(* Schneider Machine Expert - Basic project PLC1, file version 2.7.0.0 *)
(* CompanyInformations: Name=Saxion *)
(* ProjectInformations: Name=TPAC - LFT Handling *)

HARDWARE
  Cpu 0: TM221CE24T
  EthernetConfiguration: NetworkName=M221, IpAllocationMode=FixedAddress, IpAddress=10.10.120.250, SubnetMask=255.255.255.0
  SerialLineConfiguration: Baud=Baud19200, Parity=ParityEven, DataBits=DataBits8, StopBits=StopBits1, PhysicalMedium=PhysicalMediumRs485, SlaveId=1, Addressing=SlaveAddressing
  MastTask: UsePeriodScanMode=false, PeriodScan=100
  FastTask: Period=255
  CpuBehavior: StartingMode=StartAsPreviousState, AutoSaveRamOnEeprom=true, WatchdogPeriod=250

SYMBOLS  (address, symbol, comment, settings)
  %M10      ALWAYS_FALSE
  %M11      ALWAYS_TRUE
  %M20      INC_TRANSBAAN
  %M30      STAP10ACTIVEER
  %M50      B_SAFETYOK
  %M51      RUN_AUTO
  %M52      RUN_RESET
  %M53      STOP
  %M54      RUN_PRG_TEST
  %M55      RUN_PRG
  %M56      RUN_TRANSBAAN
  %M57      RUN_SIM
  %M60      KUKASTART9
  %M61      KUKASTART10
  %M62      KUKASTART11
  %M63      KUKASTART_SPARE
  %M64      KUKASTART_SPARE1
  %M65      KUKASTOP_1
  %M66      KUKASTOP_2
  %M67      KUKASTOP_3
  %M68      QX_VENTIEL1
  %M69      QX_VENTIEL2
  %M70      QX_VENTIEL3
  %M80      QX_RELAISEXSTART
  %M81      QX_RELAISEXSTOP
  %M84      QX_VENTIEL1  "Start eindbeweging"
  %M85      QX_CUTTINGTOOLACTIVEER
  %M86      QX_CUTTINGTOOLDEACTIVEER
  %M98      QX_STARTTRANSBAAN
  %M99      QX_STOPTRANSBAAN
  %M100     IX_STARTKNOP
  %M101     IX_STOPKNOP
  %M102     IX_ESTOP
  %M103     IX_FCLENGTE
  %M104     IX_FCGRIPPER
  %M105     IX_REEDCUTTINGOPEN
  %M106     IX_REEDCUTTINGGESLOTEN
  %M107     IX_REEDGRIPPER1
  %M108     IX_REEDGRIPPER2
  %M109     IX_KUKAGEREED
  %M110     IX_KUKAALARM
  %M111     IX_KUKATUSSEN
  %M112     IX_CUTTERHAND
  %M120     IX_RESET
  %MW10     PRG_STAPPEN
  %MW12     ALARMCODE_PRG
  %TM1      T_STAP1  [Preset=2, Base=OneSecond]
  %TM2      T_STAP2  [Preset=2, Base=OneSecond]
  %TM3      T_ALARMSTAP2  "Timeout voor alarm"  [Preset=60, Base=OneSecond]
  %TM4      T_ALARMSTAP4  [Preset=5, Base=OneSecond]
  %TM5      T_ALARMSTAP5  [Preset=5, Base=OneSecond]
  %TM6      T_WACHTNACUT  [Preset=2, Base=OneSecond]
  %TM7      T_ALARMSTAP7  [Preset=30, Base=OneSecond]
  %TM8      T_STAP7  [Preset=2, Base=OneSecond]
  %TM9      T_ALARMSTAP8  [Preset=10, Base=OneSecond]
  %TM10     T_STAP9  [Preset=2, Base=OneSecond]
  %TM11     T_ALARMSTAP10  [Preset=10, Base=OneSecond]
  %TM12     T_STAP10  [Type=TP, Preset=3, Base=OneSecond]
  %TM13     T_STAP11  [Preset=3, Base=OneSecond]
  %TM14     T_ALARMSTAP11  [Preset=10, Base=OneSecond]
  %TM20     T_STARTKNOP  [Preset=1, Base=OneSecond]
  %TM21     T_STOPKNOP  [Preset=1, Base=OneSecond]
  %TM66       [Preset=30, Base=OneSecond]
  %I0.0     PB01
  %I0.1     PB02
  %I0.2     PB03
  %I0.3     FC01
  %I0.4     FC02
  %I0.5     RC01
  %I0.6     RC02
  %I0.7     RG01
  %I0.8     RG02
  %I0.9     IKS01
  %I0.10    IKS02
  %I0.11    IKS03
  %I0.12    PB04

POU ALIAS
  (* SectionNumber=1 *)

// Rung 0
  LD 1                    (* Alias POU regelt in/uitgangen *)
  ST %M11                 (* ALWAYS_TRUE - Zet simuleer bit %M57 om hardware I/O inactief te zetten. *)
  STN %M10                (* ALWAYS_FALSE *)
  // as ST:
  //   ALWAYS_TRUE := TRUE;
  //   ALWAYS_FALSE := FALSE;

// Rung 1: Startknop
  BLK %TM20               (* T_STARTKNOP *)
  LD %I0.0                (* PB01 *)
  ANDN %M57               (* RUN_SIM *)
  ANDN %M120              (* IX_RESET *)
  IN
  OUT_BLK
  LD Q
  ST %M100                (* IX_STARTKNOP *)
  END_BLK
  // as ST:
  //   T_STARTKNOP(IN := PB01 AND NOT RUN_SIM AND NOT IX_RESET);
  //   IX_STARTKNOP := T_STARTKNOP.Q;

// Rung 2: Stopknop
  BLK %TM21               (* T_STOPKNOP *)
  LD %I0.1                (* PB02 *)
  ANDN %M57               (* RUN_SIM *)
  ANDN %M120              (* IX_RESET *)
  IN
  OUT_BLK
  LD Q
  ST %M101                (* IX_STOPKNOP *)
  END_BLK
  // as ST:
  //   T_STOPKNOP(IN := PB02 AND NOT RUN_SIM AND NOT IX_RESET);
  //   IX_STOPKNOP := T_STOPKNOP.Q;

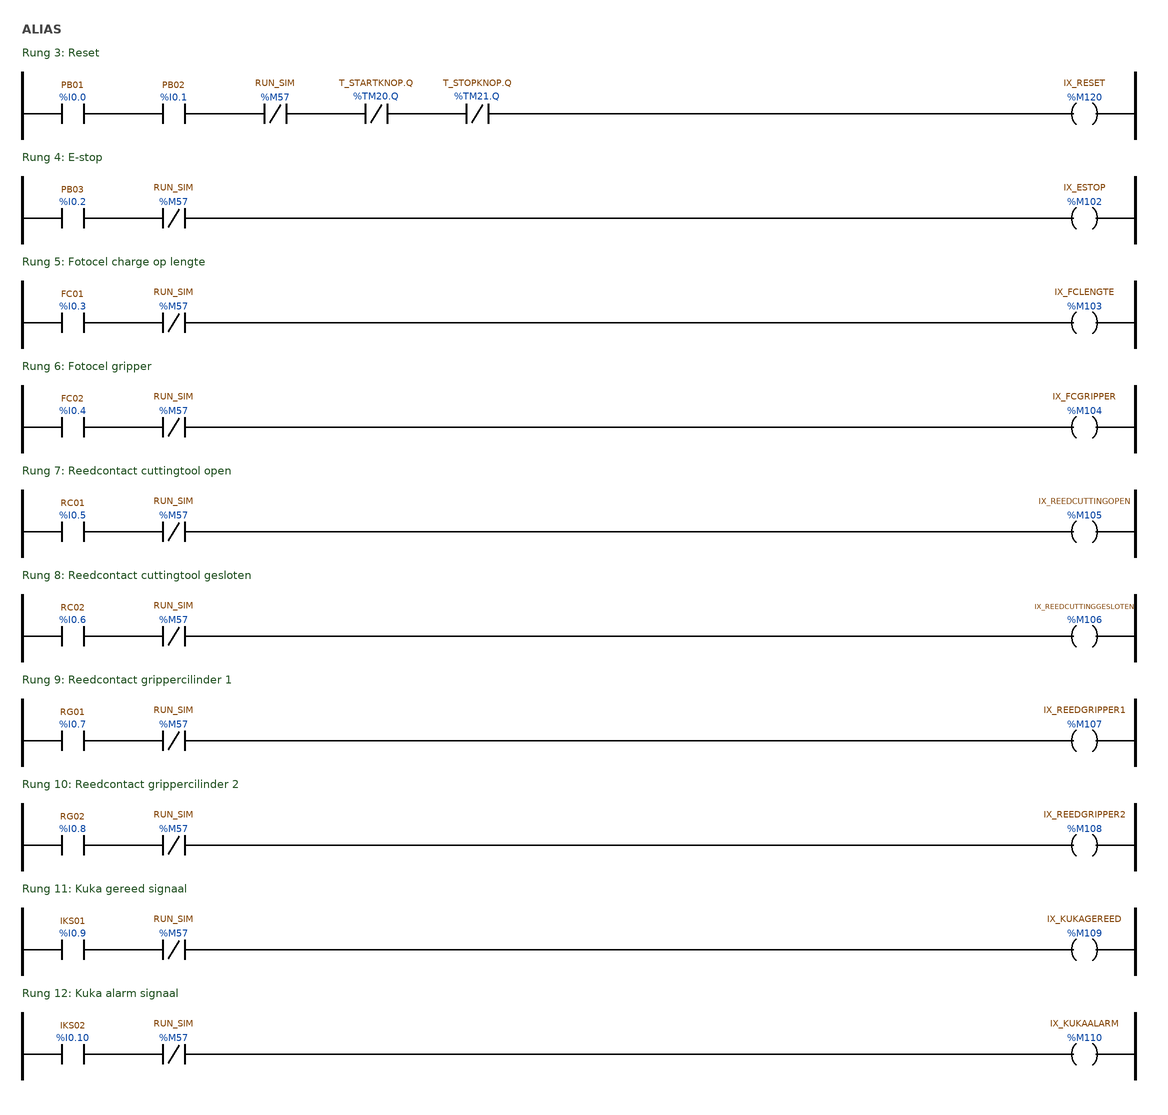

// Rung 3: Reset
  LD %I0.0                (* PB01 *)
  AND %I0.1               (* PB02 *)
  ANDN %M57               (* RUN_SIM *)
  ANDN %TM20.Q            (* T_STARTKNOP *)
  ANDN %TM21.Q            (* T_STOPKNOP *)
  ST %M120                (* IX_RESET *)
  // as ST:
  //   IX_RESET := PB01 AND PB02 AND NOT RUN_SIM AND NOT T_STARTKNOP.Q AND NOT T_STOPKNOP.Q;

// Rung 4: E-stop
  LD %I0.2                (* PB03 *)
  ANDN %M57               (* RUN_SIM *)
  ST %M102                (* IX_ESTOP *)
  // as ST:
  //   IX_ESTOP := PB03 AND NOT RUN_SIM;

// Rung 5: Fotocel charge op lengte
  LD %I0.3                (* FC01 *)
  ANDN %M57               (* RUN_SIM *)
  ST %M103                (* IX_FCLENGTE *)
  // as ST:
  //   IX_FCLENGTE := FC01 AND NOT RUN_SIM;

// Rung 6: Fotocel gripper
  LD %I0.4                (* FC02 *)
  ANDN %M57               (* RUN_SIM *)
  ST %M104                (* IX_FCGRIPPER *)
  // as ST:
  //   IX_FCGRIPPER := FC02 AND NOT RUN_SIM;

// Rung 7: Reedcontact cuttingtool open
  LD %I0.5                (* RC01 *)
  ANDN %M57               (* RUN_SIM *)
  ST %M105                (* IX_REEDCUTTINGOPEN *)
  // as ST:
  //   IX_REEDCUTTINGOPEN := RC01 AND NOT RUN_SIM;

// Rung 8: Reedcontact cuttingtool gesloten
  LD %I0.6                (* RC02 *)
  ANDN %M57               (* RUN_SIM *)
  ST %M106                (* IX_REEDCUTTINGGESLOTEN *)
  // as ST:
  //   IX_REEDCUTTINGGESLOTEN := RC02 AND NOT RUN_SIM;

// Rung 9: Reedcontact grippercilinder 1
  LD %I0.7                (* RG01 *)
  ANDN %M57               (* RUN_SIM *)
  ST %M107                (* IX_REEDGRIPPER1 *)
  // as ST:
  //   IX_REEDGRIPPER1 := RG01 AND NOT RUN_SIM;

// Rung 10: Reedcontact grippercilinder 2
  LD %I0.8                (* RG02 *)
  ANDN %M57               (* RUN_SIM *)
  ST %M108                (* IX_REEDGRIPPER2 *)
  // as ST:
  //   IX_REEDGRIPPER2 := RG02 AND NOT RUN_SIM;

// Rung 11: Kuka gereed signaal
  LD %I0.9                (* IKS01 *)
  ANDN %M57               (* RUN_SIM *)
  ST %M109                (* IX_KUKAGEREED *)
  // as ST:
  //   IX_KUKAGEREED := IKS01 AND NOT RUN_SIM;

// Rung 12: Kuka alarm signaal
  LD %I0.10               (* IKS02 *)
  ANDN %M57               (* RUN_SIM *)
  ST %M110                (* IX_KUKAALARM *)
  // as ST:
  //   IX_KUKAALARM := IKS02 AND NOT RUN_SIM;

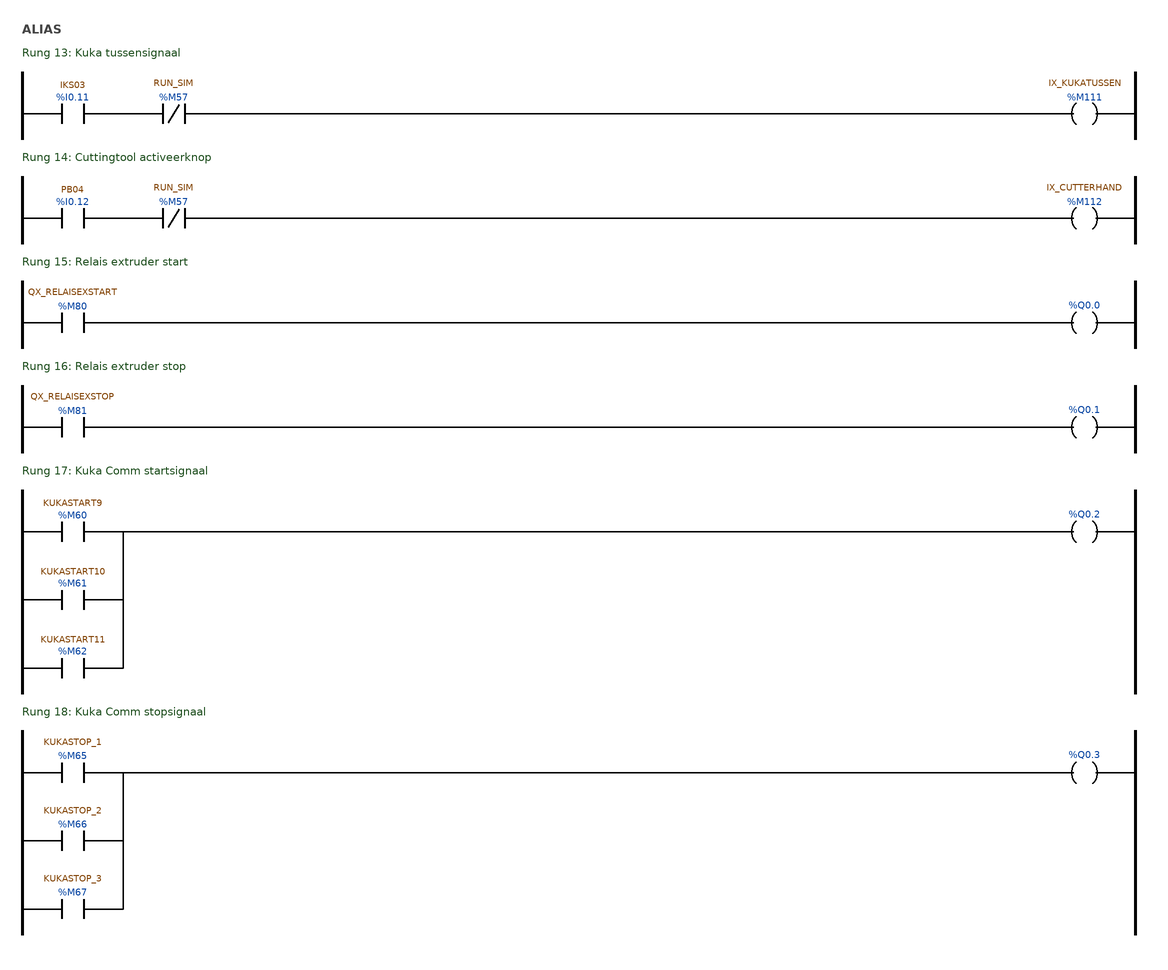

// Rung 13: Kuka tussensignaal
  LD %I0.11               (* IKS03 *)
  ANDN %M57               (* RUN_SIM *)
  ST %M111                (* IX_KUKATUSSEN *)
  // as ST:
  //   IX_KUKATUSSEN := IKS03 AND NOT RUN_SIM;

// Rung 14: Cuttingtool activeerknop
  LD %I0.12               (* PB04 *)
  ANDN %M57               (* RUN_SIM *)
  ST %M112                (* IX_CUTTERHAND *)
  // as ST:
  //   IX_CUTTERHAND := PB04 AND NOT RUN_SIM;

// Rung 15: Relais extruder start
  LD %M80                 (* QX_RELAISEXSTART *)
  ST %Q0.0
  // as ST:
  //   %Q0.0 := QX_RELAISEXSTART;

// Rung 16: Relais extruder stop
  LD %M81                 (* QX_RELAISEXSTOP *)
  ST %Q0.1
  // as ST:
  //   %Q0.1 := QX_RELAISEXSTOP;

// Rung 17: Kuka Comm startsignaal
  LD %M60                 (* KUKASTART9 *)
  OR %M61                 (* KUKASTART10 *)
  OR %M62                 (* KUKASTART11 *)
  ST %Q0.2
  // as ST:
  //   %Q0.2 := KUKASTART9 OR KUKASTART10 OR KUKASTART11;

// Rung 18: Kuka Comm stopsignaal
  LD %M65                 (* KUKASTOP_1 *)
  OR %M66                 (* KUKASTOP_2 *)
  OR %M67                 (* KUKASTOP_3 *)
  ST %Q0.3
  // as ST:
  //   %Q0.3 := KUKASTOP_1 OR KUKASTOP_2 OR KUKASTOP_3;

// Rung 19: Ventiel1/Kuka Alarmsignaal
  LD %M68                 (* QX_VENTIEL1 *)
  ST %Q0.4
  // as ST:
  //   %Q0.4 := QX_VENTIEL1;

// Rung 20
  LD %M85                 (* QX_CUTTINGTOOLACTIVEER *)
  ST %Q0.5
  // as ST:
  //   %Q0.5 := QX_CUTTINGTOOLACTIVEER;

// Rung 21
  LD %M86                 (* QX_CUTTINGTOOLDEACTIVEER *)
  ST %Q0.6
  // as ST:
  //   %Q0.6 := QX_CUTTINGTOOLDEACTIVEER;

POU Safety
  (* SectionNumber=2 *)

// Rung 22: Lees ingangen
  LD %M102                (* IX_ESTOP - // Laad E-STOP signal (NC) *)
  ANDN %M110              (* IX_KUKAALARM - // KUKA Alarm Signal (NO) *)
  ST %M50                 (* B_SAFETYOK - // Zet resultaat in safety bit *)
  // as ST:
  //   B_SAFETYOK := IX_ESTOP AND NOT IX_KUKAALARM;

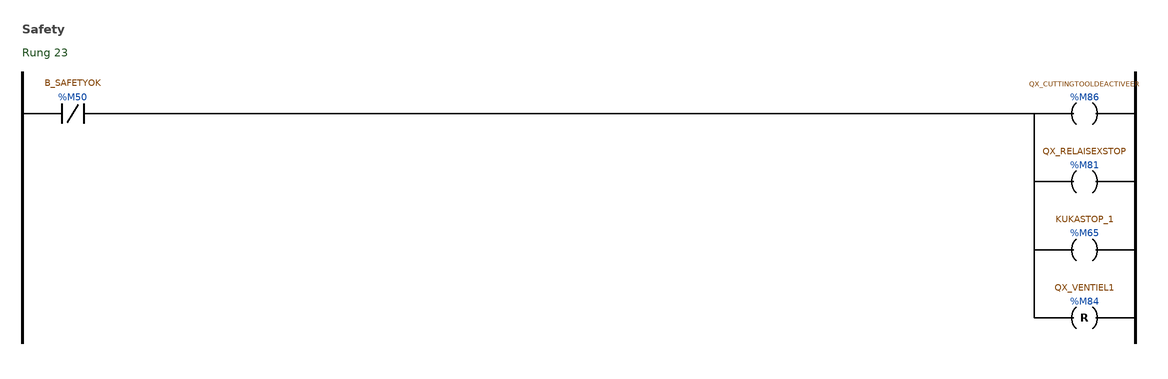

// Rung 23
  LDN %M50                (* B_SAFETYOK *)
  ST %M86                 (* QX_CUTTINGTOOLDEACTIVEER *)
  ST %M81                 (* QX_RELAISEXSTOP *)
  ST %M65                 (* KUKASTOP_1 *)
  R %M84                  (* QX_VENTIEL1 *)
  // as ST:
  //   QX_CUTTINGTOOLDEACTIVEER := NOT B_SAFETYOK;
  //   QX_RELAISEXSTOP := NOT B_SAFETYOK;
  //   KUKASTOP_1 := NOT B_SAFETYOK;
  //   IF NOT B_SAFETYOK THEN QX_VENTIEL1 := FALSE; END_IF;

POU Modus
  (* SectionNumber=3 *)

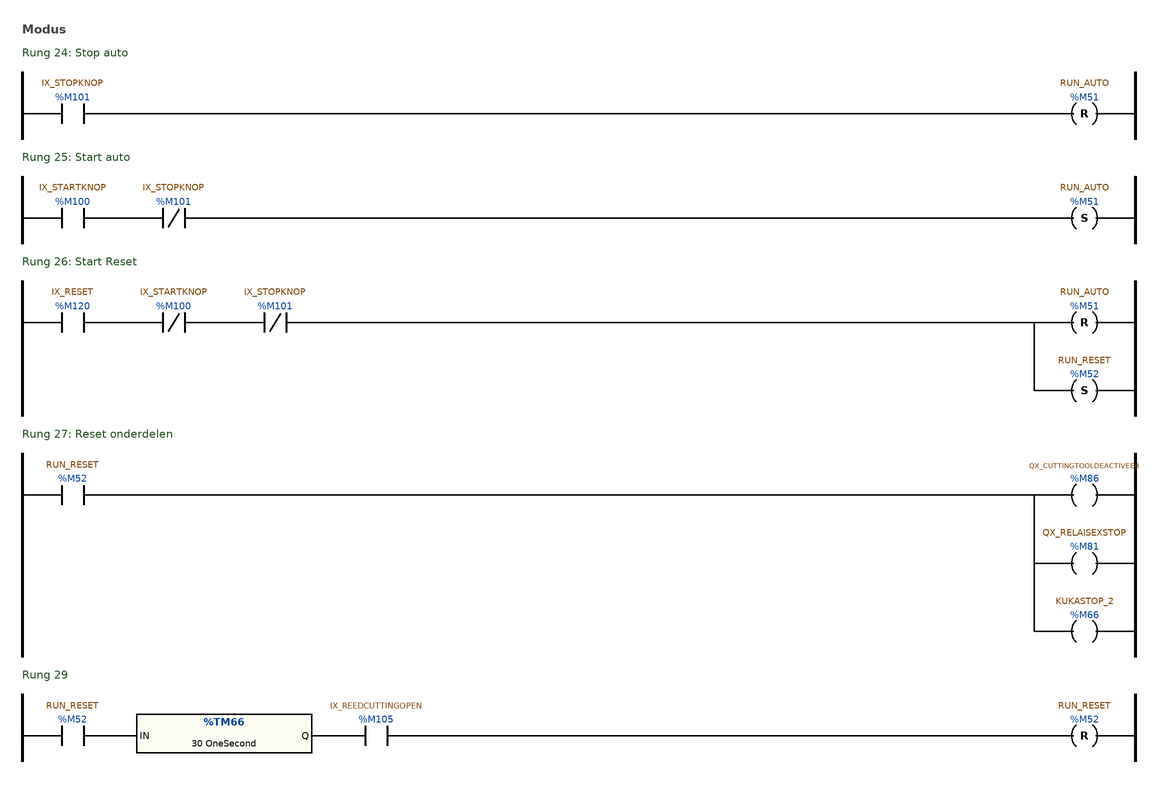

// Rung 24: Stop auto
  LD %M101                (* IX_STOPKNOP *)
  R %M51                  (* RUN_AUTO *)
  // as ST:
  //   IF IX_STOPKNOP THEN RUN_AUTO := FALSE; END_IF;

// Rung 25: Start auto
  LD %M100                (* IX_STARTKNOP *)
  ANDN %M101              (* IX_STOPKNOP *)
  S %M51                  (* RUN_AUTO *)
  // as ST:
  //   IF IX_STARTKNOP AND NOT IX_STOPKNOP THEN RUN_AUTO := TRUE; END_IF;

// Rung 26: Start Reset
  LD %M120                (* IX_RESET *)
  ANDN %M100              (* IX_STARTKNOP *)
  ANDN %M101              (* IX_STOPKNOP *)
  R %M51                  (* RUN_AUTO *)
  S %M52                  (* RUN_RESET *)
  // as ST:
  //   IF IX_RESET AND NOT IX_STARTKNOP AND NOT IX_STOPKNOP THEN RUN_AUTO := FALSE; END_IF;
  //   IF IX_RESET AND NOT IX_STARTKNOP AND NOT IX_STOPKNOP THEN RUN_RESET := TRUE; END_IF;

// Rung 27: Reset onderdelen
  LD %M52                 (* RUN_RESET *)
  ST %M86                 (* QX_CUTTINGTOOLDEACTIVEER *)
  ST %M81                 (* QX_RELAISEXSTOP *)
  ST %M66                 (* KUKASTOP_2 *)
  // as ST:
  //   QX_CUTTINGTOOLDEACTIVEER := RUN_RESET;
  //   QX_RELAISEXSTOP := RUN_RESET;
  //   KUKASTOP_2 := RUN_RESET;

// Rung 28: Reset programmastappen
// Res
  LD %M52                 (* RUN_RESET *)
  [ %MW10 := 0 ]          (* PRG_STAPPEN *)
  // as ST:
  //   IF RUN_RESET THEN PRG_STAPPEN := 0; END_IF;

// Rung 29
  BLK %TM66
  LD %M52                 (* RUN_RESET *)
  IN
  OUT_BLK
  LD Q
  AND %M105               (* IX_REEDCUTTINGOPEN *)
  R %M52                  (* RUN_RESET *)
  END_BLK
  // as ST:
  //   %TM66(IN := RUN_RESET);
  //   IF %TM66.Q AND IX_REEDCUTTINGOPEN THEN RUN_RESET := FALSE; END_IF;

POU PRG1
  (* SectionNumber=4 *)

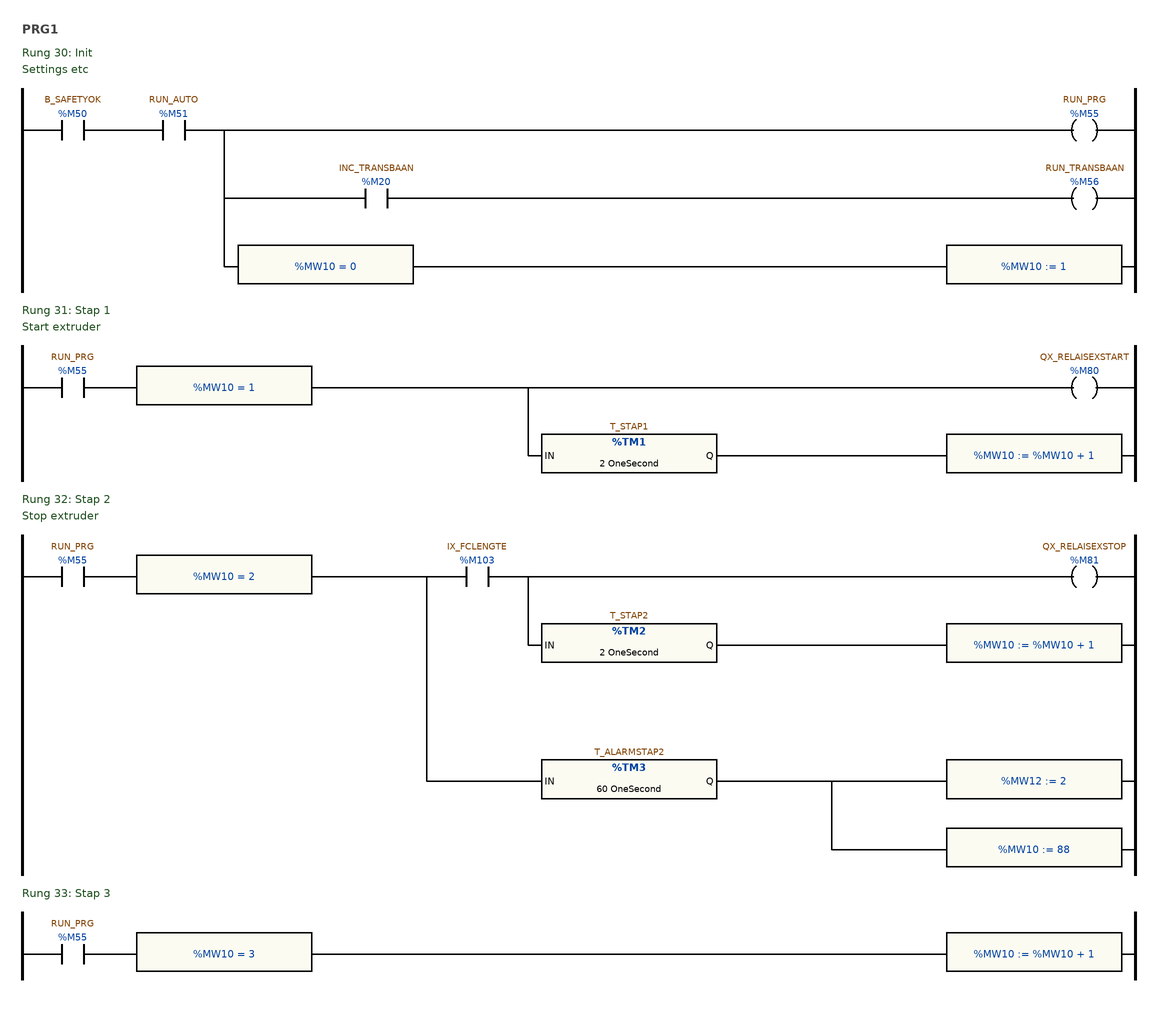

// Rung 30: Init
// Settings etc
  LD %M50                 (* B_SAFETYOK *)
  AND %M51                (* RUN_AUTO *)
  MPS
  ST %M55                 (* RUN_PRG *)
  MRD
  AND %M20                (* INC_TRANSBAAN *)
  ST %M56                 (* RUN_TRANSBAAN *)
  MPP
  AND [ %MW10 = 0 ]       (* PRG_STAPPEN *)
  [ %MW10 := 1 ]          (* PRG_STAPPEN *)
  // as ST:
  //   RUN_PRG := B_SAFETYOK AND RUN_AUTO;
  //   RUN_TRANSBAAN := B_SAFETYOK AND RUN_AUTO AND INC_TRANSBAAN;
  //   IF B_SAFETYOK AND RUN_AUTO AND PRG_STAPPEN = 0 THEN PRG_STAPPEN := 1; END_IF;

// Rung 31: Stap 1
// Start extruder
  LD 1
  MULTIFB
  LD 1
  AND %M55                (* RUN_PRG *)
  AND [ %MW10 = 1 ]       (* PRG_STAPPEN *)
  ST %MW2009:X0
  LD %MW2009:X0
  ST %M80                 (* QX_RELAISEXSTART *)
  BLK %TM1                (* T_STAP1 *)
  LD %MW2009:X0
  IN
  OUT_BLK
  LD Q
  [ %MW10 := %MW10 + 1 ]  (* PRG_STAPPEN, PRG_STAPPEN *)
  END_BLK
  MULTIFB
  // as ST:
  //   QX_RELAISEXSTART := RUN_PRG AND PRG_STAPPEN = 1;
  //   T_STAP1(IN := RUN_PRG AND PRG_STAPPEN = 1);
  //   IF T_STAP1.Q THEN PRG_STAPPEN := PRG_STAPPEN + 1; END_IF;

// Rung 32: Stap 2
// Stop extruder
  LD 1
  MULTIFB
  LD 1
  AND %M55                (* RUN_PRG *)
  AND [ %MW10 = 2 ]       (* PRG_STAPPEN *)
  ST %MW2009:X0
  LD %MW2009:X0
  AND %M103               (* IX_FCLENGTE *)
  ST %MW2009:X1
  LD %MW2009:X1
  ST %M81                 (* QX_RELAISEXSTOP *)
  BLK %TM2                (* T_STAP2 *)
  LD %MW2009:X1
  IN
  OUT_BLK
  LD Q
  [ %MW10 := %MW10 + 1 ]  (* PRG_STAPPEN, PRG_STAPPEN *)
  END_BLK
  BLK %TM3                (* T_ALARMSTAP2 *)
  LD %MW2009:X0
  IN
  OUT_BLK
  LD Q
  [ %MW12 := 2 ]          (* ALARMCODE_PRG *)
  [ %MW10 := 88 ]         (* PRG_STAPPEN *)
  END_BLK
  MULTIFB
  // as ST:
  //   QX_RELAISEXSTOP := RUN_PRG AND PRG_STAPPEN = 2 AND IX_FCLENGTE;
  //   T_STAP2(IN := RUN_PRG AND PRG_STAPPEN = 2 AND IX_FCLENGTE);
  //   _t1 := RUN_PRG AND PRG_STAPPEN = 2;
  //   IF T_STAP2.Q THEN PRG_STAPPEN := PRG_STAPPEN + 1; END_IF;
  //   T_ALARMSTAP2(IN := _t1);
  //   IF T_ALARMSTAP2.Q THEN ALARMCODE_PRG := 2; END_IF;
  //   IF T_ALARMSTAP2.Q THEN PRG_STAPPEN := 88; END_IF;

// Rung 33: Stap 3
  LD %M55                 (* RUN_PRG *)
  AND [ %MW10 = 3 ]       (* PRG_STAPPEN *)
  [ %MW10 := %MW10 + 1 ]  (* PRG_STAPPEN, PRG_STAPPEN *)
  // as ST:
  //   IF RUN_PRG AND PRG_STAPPEN = 3 THEN PRG_STAPPEN := PRG_STAPPEN + 1; END_IF;

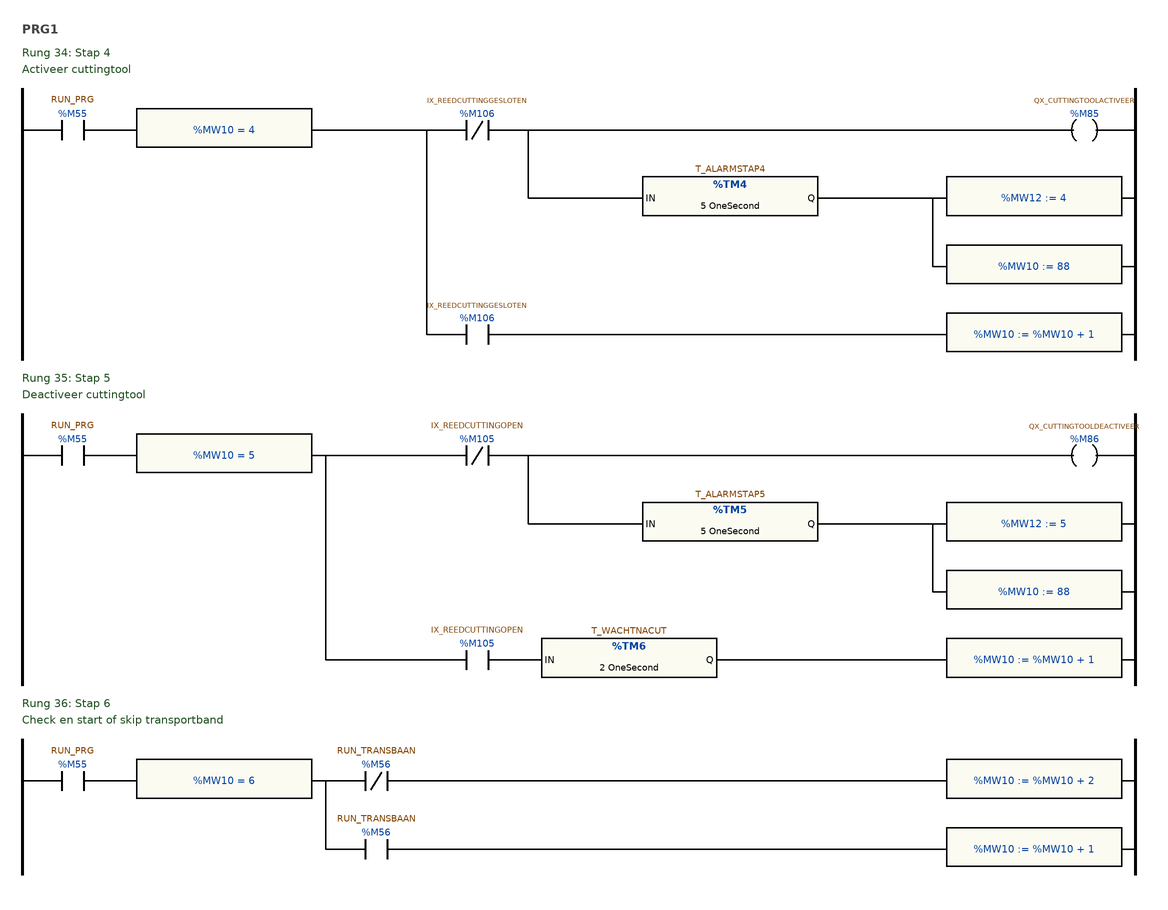

// Rung 34: Stap 4
// Activeer cuttingtool
  LD 1
  MULTIFB
  LD 1
  AND %M55                (* RUN_PRG *)
  AND [ %MW10 = 4 ]       (* PRG_STAPPEN *)
  ST %MW2009:X0
  LD %MW2009:X0
  ANDN %M106              (* IX_REEDCUTTINGGESLOTEN *)
  ST %MW2009:X1
  LD %MW2009:X1
  ST %M85                 (* QX_CUTTINGTOOLACTIVEER *)
  BLK %TM4                (* T_ALARMSTAP4 *)
  LD %MW2009:X1
  IN
  OUT_BLK
  LD Q
  [ %MW12 := 4 ]          (* ALARMCODE_PRG *)
  [ %MW10 := 88 ]         (* PRG_STAPPEN *)
  END_BLK
  LD %MW2009:X0
  AND %M106               (* IX_REEDCUTTINGGESLOTEN *)
  [ %MW10 := %MW10 + 1 ]  (* PRG_STAPPEN, PRG_STAPPEN *)
  MULTIFB
  // as ST:
  //   QX_CUTTINGTOOLACTIVEER := RUN_PRG AND PRG_STAPPEN = 4 AND NOT IX_REEDCUTTINGGESLOTEN;
  //   T_ALARMSTAP4(IN := RUN_PRG AND PRG_STAPPEN = 4 AND NOT IX_REEDCUTTINGGESLOTEN);
  //   IF T_ALARMSTAP4.Q THEN ALARMCODE_PRG := 4; END_IF;
  //   _t1 := RUN_PRG AND PRG_STAPPEN = 4;
  //   IF T_ALARMSTAP4.Q THEN PRG_STAPPEN := 88; END_IF;
  //   IF _t1 AND IX_REEDCUTTINGGESLOTEN THEN PRG_STAPPEN := PRG_STAPPEN + 1; END_IF;

// Rung 35: Stap 5
// Deactiveer cuttingtool
  LD 1
  MULTIFB
  LD 1
  AND %M55                (* RUN_PRG *)
  AND [ %MW10 = 5 ]       (* PRG_STAPPEN *)
  ST %MW2009:X0
  LD %MW2009:X0
  ANDN %M105              (* IX_REEDCUTTINGOPEN *)
  ST %MW2009:X1
  LD %MW2009:X1
  ST %M86                 (* QX_CUTTINGTOOLDEACTIVEER *)
  BLK %TM5                (* T_ALARMSTAP5 *)
  LD %MW2009:X1
  IN
  OUT_BLK
  LD Q
  [ %MW12 := 5 ]          (* ALARMCODE_PRG *)
  [ %MW10 := 88 ]         (* PRG_STAPPEN *)
  END_BLK
  BLK %TM6                (* T_WACHTNACUT *)
  LD %MW2009:X0
  AND %M105               (* IX_REEDCUTTINGOPEN *)
  IN
  OUT_BLK
  LD Q
  [ %MW10 := %MW10 + 1 ]  (* PRG_STAPPEN, PRG_STAPPEN *)
  END_BLK
  MULTIFB
  // as ST:
  //   QX_CUTTINGTOOLDEACTIVEER := RUN_PRG AND PRG_STAPPEN = 5 AND NOT IX_REEDCUTTINGOPEN;
  //   T_ALARMSTAP5(IN := RUN_PRG AND PRG_STAPPEN = 5 AND NOT IX_REEDCUTTINGOPEN);
  //   IF T_ALARMSTAP5.Q THEN ALARMCODE_PRG := 5; END_IF;
  //   _t1 := RUN_PRG AND PRG_STAPPEN = 5;
  //   IF T_ALARMSTAP5.Q THEN PRG_STAPPEN := 88; END_IF;
  //   T_WACHTNACUT(IN := _t1 AND IX_REEDCUTTINGOPEN);
  //   IF T_WACHTNACUT.Q THEN PRG_STAPPEN := PRG_STAPPEN + 1; END_IF;

// Rung 36: Stap 6
// Check en start of skip transportband
  LD %M55                 (* RUN_PRG *)
  AND [ %MW10 = 6 ]       (* PRG_STAPPEN *)
  MPS
  ANDN %M56               (* RUN_TRANSBAAN *)
  [ %MW10 := %MW10 + 2 ]  (* PRG_STAPPEN, PRG_STAPPEN *)
  MPP
  AND %M56                (* RUN_TRANSBAAN *)
  [ %MW10 := %MW10 + 1 ]  (* PRG_STAPPEN, PRG_STAPPEN *)
  // as ST:
  //   _t1 := RUN_PRG AND PRG_STAPPEN = 6;
  //   IF RUN_PRG AND PRG_STAPPEN = 6 AND NOT RUN_TRANSBAAN THEN PRG_STAPPEN := PRG_STAPPEN + 2; END_IF;
  //   IF _t1 AND RUN_TRANSBAAN THEN PRG_STAPPEN := PRG_STAPPEN + 1; END_IF;

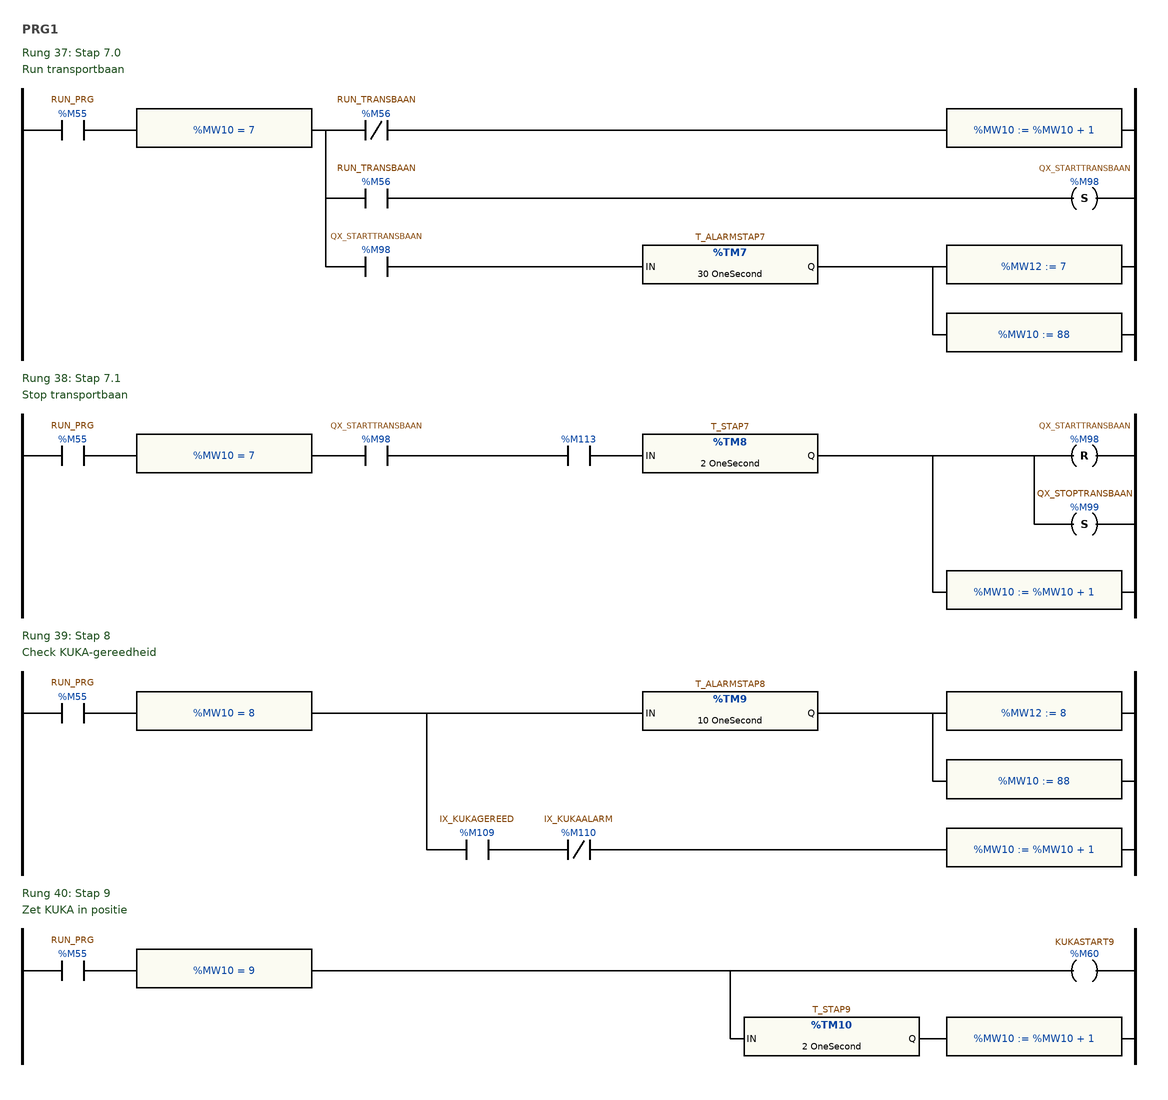

// Rung 37: Stap 7.0
// Run transportbaan
  LD 1
  MULTIFB
  LD 1
  AND %M55                (* RUN_PRG *)
  AND [ %MW10 = 7 ]       (* PRG_STAPPEN *)
  ST %MW2009:X0
  LD %MW2009:X0
  MPS
  ANDN %M56               (* RUN_TRANSBAAN *)
  [ %MW10 := %MW10 + 1 ]  (* PRG_STAPPEN, PRG_STAPPEN *)
  MPP
  AND %M56                (* RUN_TRANSBAAN *)
  S %M98                  (* QX_STARTTRANSBAAN *)
  BLK %TM7                (* T_ALARMSTAP7 *)
  LD %MW2009:X0
  AND %M98                (* QX_STARTTRANSBAAN *)
  IN
  OUT_BLK
  LD Q
  [ %MW12 := 7 ]          (* ALARMCODE_PRG *)
  [ %MW10 := 88 ]         (* PRG_STAPPEN *)
  END_BLK
  MULTIFB
  // as ST:
  //   _t1 := RUN_PRG AND PRG_STAPPEN = 7;
  //   IF RUN_PRG AND PRG_STAPPEN = 7 AND NOT RUN_TRANSBAAN THEN PRG_STAPPEN := PRG_STAPPEN + 1; END_IF;
  //   IF _t1 AND RUN_TRANSBAAN THEN QX_STARTTRANSBAAN := TRUE; END_IF;
  //   T_ALARMSTAP7(IN := _t1 AND QX_STARTTRANSBAAN);
  //   IF T_ALARMSTAP7.Q THEN ALARMCODE_PRG := 7; END_IF;
  //   IF T_ALARMSTAP7.Q THEN PRG_STAPPEN := 88; END_IF;

// Rung 38: Stap 7.1
// Stop transportbaan
  BLK %TM8                (* T_STAP7 *)
  LD %M55                 (* RUN_PRG *)
  AND [ %MW10 = 7 ]       (* PRG_STAPPEN *)
  AND %M98                (* QX_STARTTRANSBAAN *)
  AND %M113
  IN
  OUT_BLK
  LD Q
  R %M98                  (* QX_STARTTRANSBAAN *)
  S %M99                  (* QX_STOPTRANSBAAN *)
  [ %MW10 := %MW10 + 1 ]  (* PRG_STAPPEN, PRG_STAPPEN *)
  END_BLK
  // as ST:
  //   T_STAP7(IN := RUN_PRG AND PRG_STAPPEN = 7 AND QX_STARTTRANSBAAN AND %M113);
  //   IF T_STAP7.Q THEN QX_STARTTRANSBAAN := FALSE; END_IF;
  //   IF T_STAP7.Q THEN QX_STOPTRANSBAAN := TRUE; END_IF;
  //   IF T_STAP7.Q THEN PRG_STAPPEN := PRG_STAPPEN + 1; END_IF;

// Rung 39: Stap 8
// Check KUKA-gereedheid
  LD 1
  MULTIFB
  LD 1
  AND %M55                (* RUN_PRG *)
  AND [ %MW10 = 8 ]       (* PRG_STAPPEN *)
  ST %MW2009:X0
  BLK %TM9                (* T_ALARMSTAP8 *)
  LD %MW2009:X0
  IN
  OUT_BLK
  LD Q
  [ %MW12 := 8 ]          (* ALARMCODE_PRG *)
  [ %MW10 := 88 ]         (* PRG_STAPPEN *)
  END_BLK
  LD %MW2009:X0
  AND %M109               (* IX_KUKAGEREED *)
  ANDN %M110              (* IX_KUKAALARM *)
  [ %MW10 := %MW10 + 1 ]  (* PRG_STAPPEN, PRG_STAPPEN *)
  MULTIFB
  // as ST:
  //   T_ALARMSTAP8(IN := RUN_PRG AND PRG_STAPPEN = 8);
  //   IF T_ALARMSTAP8.Q THEN ALARMCODE_PRG := 8; END_IF;
  //   _t1 := RUN_PRG AND PRG_STAPPEN = 8;
  //   IF T_ALARMSTAP8.Q THEN PRG_STAPPEN := 88; END_IF;
  //   IF _t1 AND IX_KUKAGEREED AND NOT IX_KUKAALARM THEN PRG_STAPPEN := PRG_STAPPEN + 1; END_IF;

// Rung 40: Stap 9
// Zet KUKA in positie
  LD 1
  MULTIFB
  LD 1
  AND %M55                (* RUN_PRG *)
  AND [ %MW10 = 9 ]       (* PRG_STAPPEN *)
  ST %MW2009:X0
  LD %MW2009:X0
  ST %M60                 (* KUKASTART9 *)
  BLK %TM10               (* T_STAP9 *)
  LD %MW2009:X0
  IN
  OUT_BLK
  LD Q
  [ %MW10 := %MW10 + 1 ]  (* PRG_STAPPEN, PRG_STAPPEN *)
  END_BLK
  MULTIFB
  // as ST:
  //   KUKASTART9 := RUN_PRG AND PRG_STAPPEN = 9;
  //   T_STAP9(IN := RUN_PRG AND PRG_STAPPEN = 9);
  //   IF T_STAP9.Q THEN PRG_STAPPEN := PRG_STAPPEN + 1; END_IF;

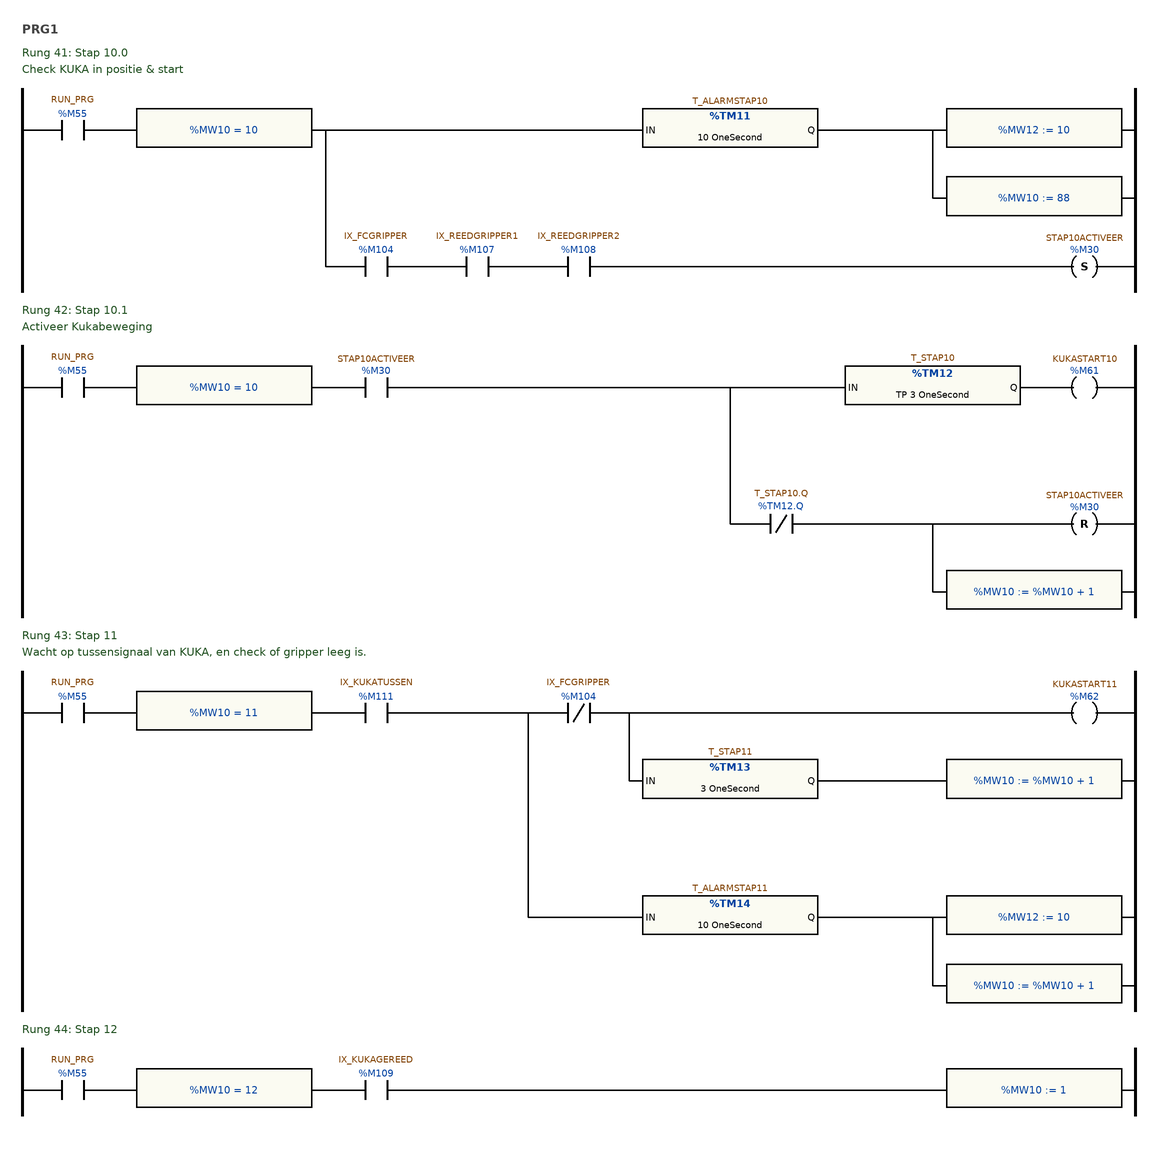

// Rung 41: Stap 10.0
// Check KUKA in positie & start
  LD 1
  MULTIFB
  LD 1
  AND %M55                (* RUN_PRG *)
  AND [ %MW10 = 10 ]      (* PRG_STAPPEN *)
  ST %MW2009:X0
  BLK %TM11               (* T_ALARMSTAP10 *)
  LD %MW2009:X0
  IN
  OUT_BLK
  LD Q
  [ %MW12 := 10 ]         (* ALARMCODE_PRG *)
  [ %MW10 := 88 ]         (* PRG_STAPPEN *)
  END_BLK
  LD %MW2009:X0
  AND %M104               (* IX_FCGRIPPER *)
  AND %M107               (* IX_REEDGRIPPER1 *)
  AND %M108               (* IX_REEDGRIPPER2 *)
  S %M30                  (* STAP10ACTIVEER *)
  MULTIFB
  // as ST:
  //   T_ALARMSTAP10(IN := RUN_PRG AND PRG_STAPPEN = 10);
  //   IF T_ALARMSTAP10.Q THEN ALARMCODE_PRG := 10; END_IF;
  //   _t1 := RUN_PRG AND PRG_STAPPEN = 10;
  //   IF T_ALARMSTAP10.Q THEN PRG_STAPPEN := 88; END_IF;
  //   IF _t1 AND IX_FCGRIPPER AND IX_REEDGRIPPER1 AND IX_REEDGRIPPER2 THEN STAP10ACTIVEER := TRUE; END_IF;

// Rung 42: Stap 10.1
// Activeer Kukabeweging
  LD 1
  MULTIFB
  LD 1
  AND %M55                (* RUN_PRG *)
  AND [ %MW10 = 10 ]      (* PRG_STAPPEN *)
  AND %M30                (* STAP10ACTIVEER *)
  ST %MW2009:X0
  BLK %TM12               (* T_STAP10 *)
  LD %MW2009:X0
  IN
  OUT_BLK
  LD Q
  ST %M61                 (* KUKASTART10 *)
  END_BLK
  LD %MW2009:X0
  ANDN %TM12.Q            (* T_STAP10 *)
  R %M30                  (* STAP10ACTIVEER *)
  [ %MW10 := %MW10 + 1 ]  (* PRG_STAPPEN, PRG_STAPPEN *)
  MULTIFB
  // as ST:
  //   T_STAP10(IN := RUN_PRG AND PRG_STAPPEN = 10 AND STAP10ACTIVEER);
  //   KUKASTART10 := T_STAP10.Q;
  //   _t1 := RUN_PRG AND PRG_STAPPEN = 10 AND STAP10ACTIVEER AND NOT T_STAP10.Q;
  //   IF _t1 THEN STAP10ACTIVEER := FALSE; END_IF;
  //   IF _t1 THEN PRG_STAPPEN := PRG_STAPPEN + 1; END_IF;

// Rung 43: Stap 11
// Wacht op tussensignaal van KUKA, en check of gripper leeg is.
  LD 1
  MULTIFB
  LD 1
  AND %M55                (* RUN_PRG *)
  AND [ %MW10 = 11 ]      (* PRG_STAPPEN *)
  AND %M111               (* IX_KUKATUSSEN *)
  ST %MW2009:X0
  LD %MW2009:X0
  ANDN %M104              (* IX_FCGRIPPER *)
  ST %MW2009:X1
  LD %MW2009:X1
  ST %M62                 (* KUKASTART11 *)
  BLK %TM13               (* T_STAP11 *)
  LD %MW2009:X1
  IN
  OUT_BLK
  LD Q
  [ %MW10 := %MW10 + 1 ]  (* PRG_STAPPEN, PRG_STAPPEN *)
  END_BLK
  BLK %TM14               (* T_ALARMSTAP11 *)
  LD %MW2009:X0
  IN
  OUT_BLK
  LD Q
  [ %MW12 := 10 ]         (* ALARMCODE_PRG *)
  [ %MW10 := %MW10 + 1 ]  (* PRG_STAPPEN, PRG_STAPPEN *)
  END_BLK
  MULTIFB
  // as ST:
  //   KUKASTART11 := RUN_PRG AND PRG_STAPPEN = 11 AND IX_KUKATUSSEN AND NOT IX_FCGRIPPER;
  //   T_STAP11(IN := RUN_PRG AND PRG_STAPPEN = 11 AND IX_KUKATUSSEN AND NOT IX_FCGRIPPER);
  //   _t1 := RUN_PRG AND PRG_STAPPEN = 11 AND IX_KUKATUSSEN;
  //   IF T_STAP11.Q THEN PRG_STAPPEN := PRG_STAPPEN + 1; END_IF;
  //   T_ALARMSTAP11(IN := _t1);
  //   IF T_ALARMSTAP11.Q THEN ALARMCODE_PRG := 10; END_IF;
  //   IF T_ALARMSTAP11.Q THEN PRG_STAPPEN := PRG_STAPPEN + 1; END_IF;

// Rung 44: Stap 12
  LD %M55                 (* RUN_PRG *)
  AND [ %MW10 = 12 ]      (* PRG_STAPPEN *)
  AND %M109               (* IX_KUKAGEREED *)
  [ %MW10 := 1 ]          (* PRG_STAPPEN *)
  // as ST:
  //   IF RUN_PRG AND PRG_STAPPEN = 12 AND IX_KUKAGEREED THEN PRG_STAPPEN := 1; END_IF;

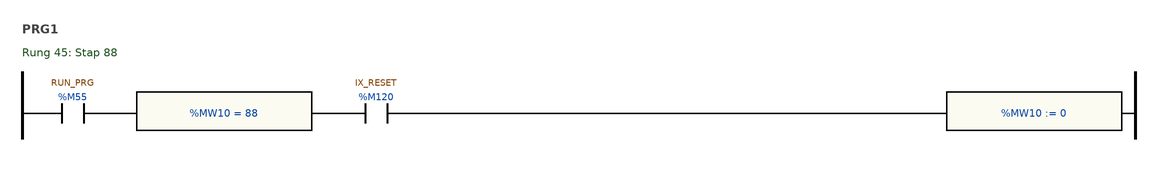

// Rung 45: Stap 88
  LD %M55                 (* RUN_PRG *)
  AND [ %MW10 = 88 ]      (* PRG_STAPPEN *)
  AND %M120               (* IX_RESET *)
  [ %MW10 := 0 ]          (* PRG_STAPPEN *)
  // as ST:
  //   IF RUN_PRG AND PRG_STAPPEN = 88 AND IX_RESET THEN PRG_STAPPEN := 0; END_IF;
